// Mitsubishi GX Works2 project: PLC응용기말고사프로젝트   PLC: Q03UDE

PROGRAM MAIN
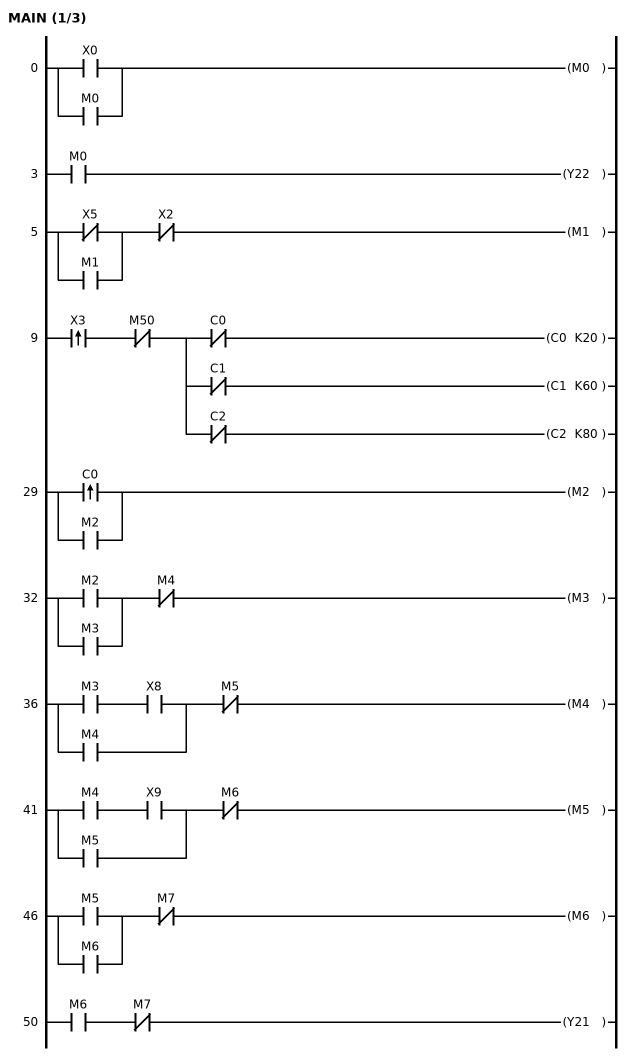
0     LD      X0
      OR      M0
      OUT     M0
3     LD      M0
      OUT     Y22
5     LDI     X5
      OR      M1
      ANI     X2
      OUT     M1
9     LDP     X3
      ANI     M50
      MPS
      ANI     C0
      OUT     C0 K20
      MRD
      ANI     C1
      OUT     C1 K60
      MPP
      ANI     C2
      OUT     C2 K80
29    LDP     C0
      OR      M2
      OUT     M2
32    LD      M2
      OR      M3
      ANI     M4
      OUT     M3
36    LD      M3
      AND     X8
      OR      M4
      ANI     M5
      OUT     M4
41    LD      M4
      AND     X9
      OR      M5
      ANI     M6
      OUT     M5
46    LD      M5
      OR      M6
      ANI     M7
      OUT     M6
50    LD      M6
      ANI     M7
      OUT     Y21
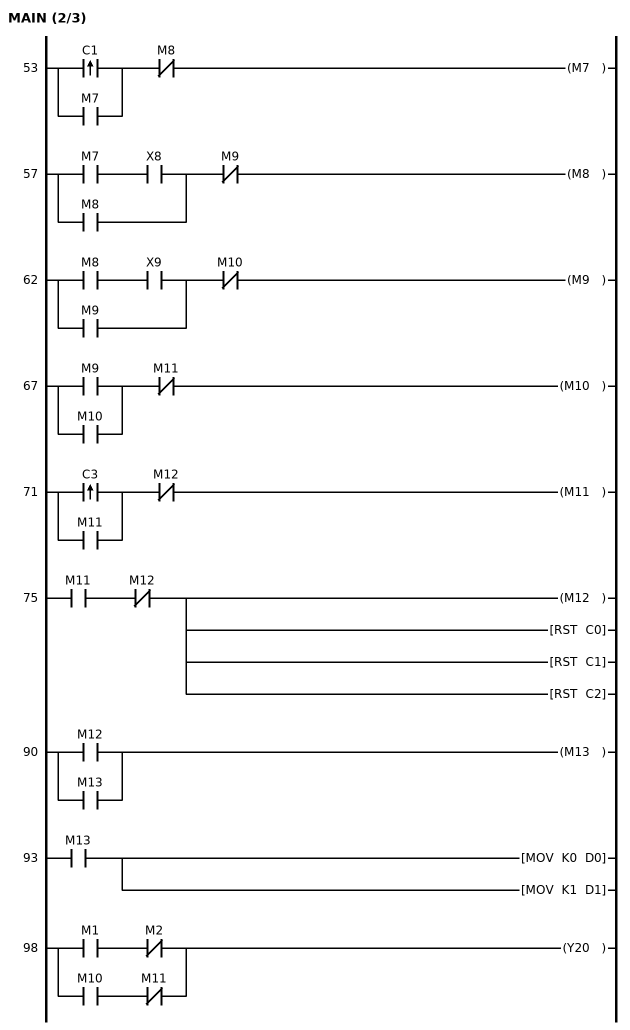
53    LDP     C1
      OR      M7
      ANI     M8
      OUT     M7
57    LD      M7
      AND     X8
      OR      M8
      ANI     M9
      OUT     M8
62    LD      M8
      AND     X9
      OR      M9
      ANI     M10
      OUT     M9
67    LD      M9
      OR      M10
      ANI     M11
      OUT     M10
71    LDP     C3
      OR      M11
      ANI     M12
      OUT     M11
75    LD      M11
      ANI     M12
      OUT     M12
      RST     C0
      RST     C1
      RST     C2
90    LD      M12
      OR      M13
      OUT     M13
93    LD      M13
      MOV     K0 D0
      MOV     K1 D1
98    LD      M1
      ANI     M2
      LD      M10
      ANI     M11
      ORB
      OUT     Y20
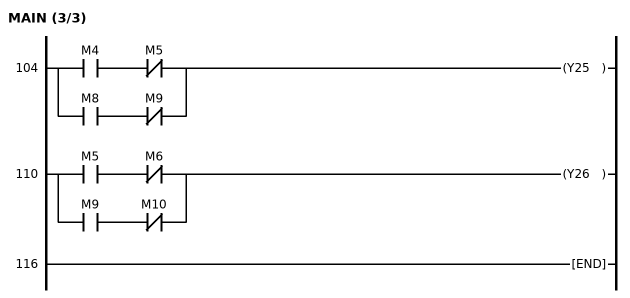
104   LD      M4
      ANI     M5
      LD      M8
      ANI     M9
      ORB
      OUT     Y25
110   LD      M5
      ANI     M6
      LD      M9
      ANI     M10
      ORB
      OUT     Y26
116   END
END_PROGRAM
